FUNCTION rotX : mat3d
VAR_INPUT
	i_ang : LREAL;
END_VAR
VAR
	rot :Mat3d := g_eye3d;
END_VAR

rot[2,2]:=COS(i_ang);
rot[3,3]:=rot[2,2];
rot[3,2]:=SIN(i_ang);
rot[2,3]:=-rot[3,2];
rotX :=rot;

END_FUNCTION

(* stored: Version 1.1.0.1, ProductVersion 3.1.4024.11
   POU rotX: Id {e7448ad1-988f-46ca-886a-6ce44eea6109}, SpecialFunc None *)
